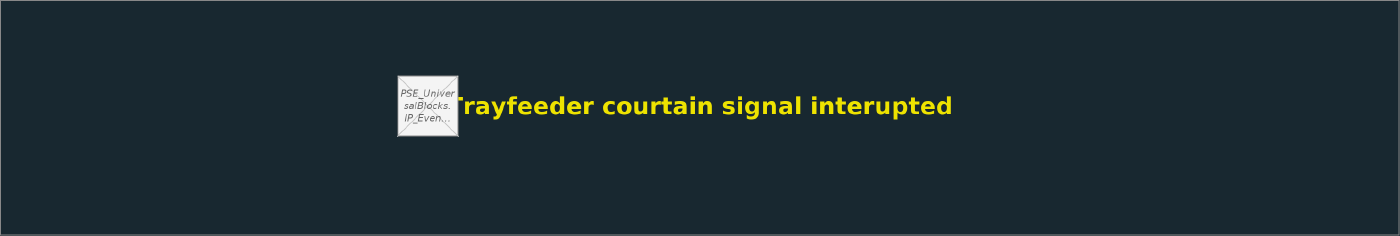
VISUALIZATION InitializingTrayfeederCourtainBroken  // 1480x250
    Label (0,92 1480x40), "Trayfeeder courtain signal interupted"
    Image (420,80 64x64), image: PSE_UniversalBlocks.IP_EventSeverity.error
END_VISUALIZATION

(* stored: Version 1.1.0.1, ProductVersion 3.1.4024.9
   Visu InitializingTrayfeederCourtainBroken: Id {a106f3ea-4f3f-4c8f-ad6d-be997126d0bd} *)
